Fanuc KAREL source: SET_PORT_ATR.kl

PROGRAM T
%NOLOCKGROUP
VAR
 v0 : INTEGER
 v1 : INTEGER
 v2 : INTEGER
 res : INTEGER
BEGIN
 res = SET_PORT_ATR(v0, v1, v2)
END T
